VAR_GLOBAL


	tPhCurrent					: REAL := 0.0;
	tPhLastReadingValid			: BOOL := FALSE;
	tOrpCurrent					: REAL := 0.0;
	tOrpLastReadingValid		: BOOL := FALSE;


	(* temperature control *)
	pumpOn				AT %Q* 	: BOOL := FALSE;
	coldValve			AT %Q* 	: BOOL := FALSE;
	hotValve			AT %Q* 	: BOOL := FALSE;
	steriValve			AT %Q*	: BOOL := FALSE; 
	//
	pwmDutyCycle				: REAL := 0.0;	
	
	jacketTempRaw		AT %I*	: INT;
	jacketTempC					: REAL := 0.0;
	jacketTempK					: REAL := 0.0;
	
	
	tempControlStop				: BOOL := FALSE;
	tempControlStart			: BOOL := FALSE;
	hotValveButton				: BOOL := FALSE;
	coldValveButton				: BOOL := FALSE;
	
	pumpIsRunning				: BOOL := FALSE;
	tempControlRunning			: BOOL := FALSE;
	tempSafetyEnabled			: BOOL := FALSE;
	
	steriStart					: BOOL := FALSE;
	steriStop					: BOOL := FALSE;
	steriRunning				: BOOL := FALSE;

	
	currentMeanTemp				: REAL := 0;
	currentTempValid			: BOOL := FALSE;
	(* target temp -> see retains *) 
	
	tempIsBelowSteriTemp		: BOOL := TRUE;
	(* target steri temp --> see retains *)	

	
END_VAR

VAR_GLOBAL PERSISTENT
	targetControlTemp			: REAL;
	targetSteriTemp				: REAL;
	targetSteriTimeMinutes		: INT;
	remainingSteriTimeMinutes	: REAL;
	
	
	remainingSteriTimeInMs		: DINT; (* 30 min in ms *)
	
	countTempSpikes				: INT;
	countValveMaxTimeExceeded	: INT;

	pidResetCounter				: INT;
END_VAR

VAR_GLOBAL CONSTANT
	CYCLE_TIME_IN_MS		: TIME := T#10ms;
END_VAR

(* stored: Version 1.1.0.1, ProductVersion 3.1.4022.12
   GVL GVL_TemperatureControl: Id {92f0593a-90ab-4fcc-a23e-30239ee482b5} *)
